(*
A. Wallace 2019-4-22
The photon energy watcher ensures the current and target photon energy is within
the arbirated bounds. Target in this case means, the calculated target photon energy
from the PVs that control the mechatronics of the undulators/ the electron energy.

If there are control PVs that match the monitor PVs, the control PVs are used to 
calculate a "target" photon energy. This is supposed to cover when the undulators/
electron energy is transitioning.

The abritrated bounds come from a simple AND of all the permitted ranges. See
the arbitrate action of the arbiter FB.

Note, this protection logic does not account for beam-off when determining fast-fault
status. If a device is requesting a limited range of eV, this request must be honored,
regardless of current beam-rate.
*)
FUNCTION_BLOCK FB_PhotonEnergyWatcher
VAR_INPUT
	i_stCurrentBeamParams	:	ST_BeamParams; //Link to global beam params
	i_stMachineTargetBeamParams	:	ST_BeamParams; //Link to global machine target beam params
	i_stRequestedBeamParams	:	ST_BeamParams; //Link to arbiter output or beam param. requestor
	// Reset fault
	i_xReset: BOOL;
END_VAR
VAR_OUTPUT
END_VAR
VAR_IN_OUT
	io_fbFFHWO	:	FB_HardwareFFOutput;
END_VAR
VAR
	xPhotonEnergyWithinBounds	:	BOOL;
	fbFF	:	FB_FastFault;
END_VAR

xPhotonEnergyWithinBounds := (i_stCurrentBeamParams.neVRange AND i_stRequestedBeamParams.neVRange) = i_stCurrentBeamParams.neVRange;

fbFF(i_xOK := xPhotonEnergyWithinBounds,
	i_xReset := i_xReset,
	io_fbFFHWO := io_fbFFHWO);

END_FUNCTION_BLOCK

(* stored: Version 1.1.0.1, ProductVersion 3.1.4024.0
   POU FB_PhotonEnergyWatcher: Id {dedd735b-7eee-031d-1b56-a60d5aa8ea22}, SpecialFunc None *)
